FUNCTION_BLOCK conveyor
  (* Standard: 61499-2 *)
  (* Version 0.1, 2017-00-25, hpea485, UOA *)
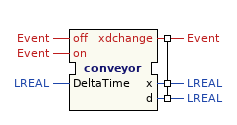
  EVENT_INPUT
    off;
    on;
  END_EVENT
  EVENT_OUTPUT
    xdchange WITH x, d;
  END_EVENT
  VAR_INPUT
    DeltaTime : LREAL := 0.01;
  END_VAR
  VAR_OUTPUT
    x : LREAL;
    d : LREAL;
  END_VAR
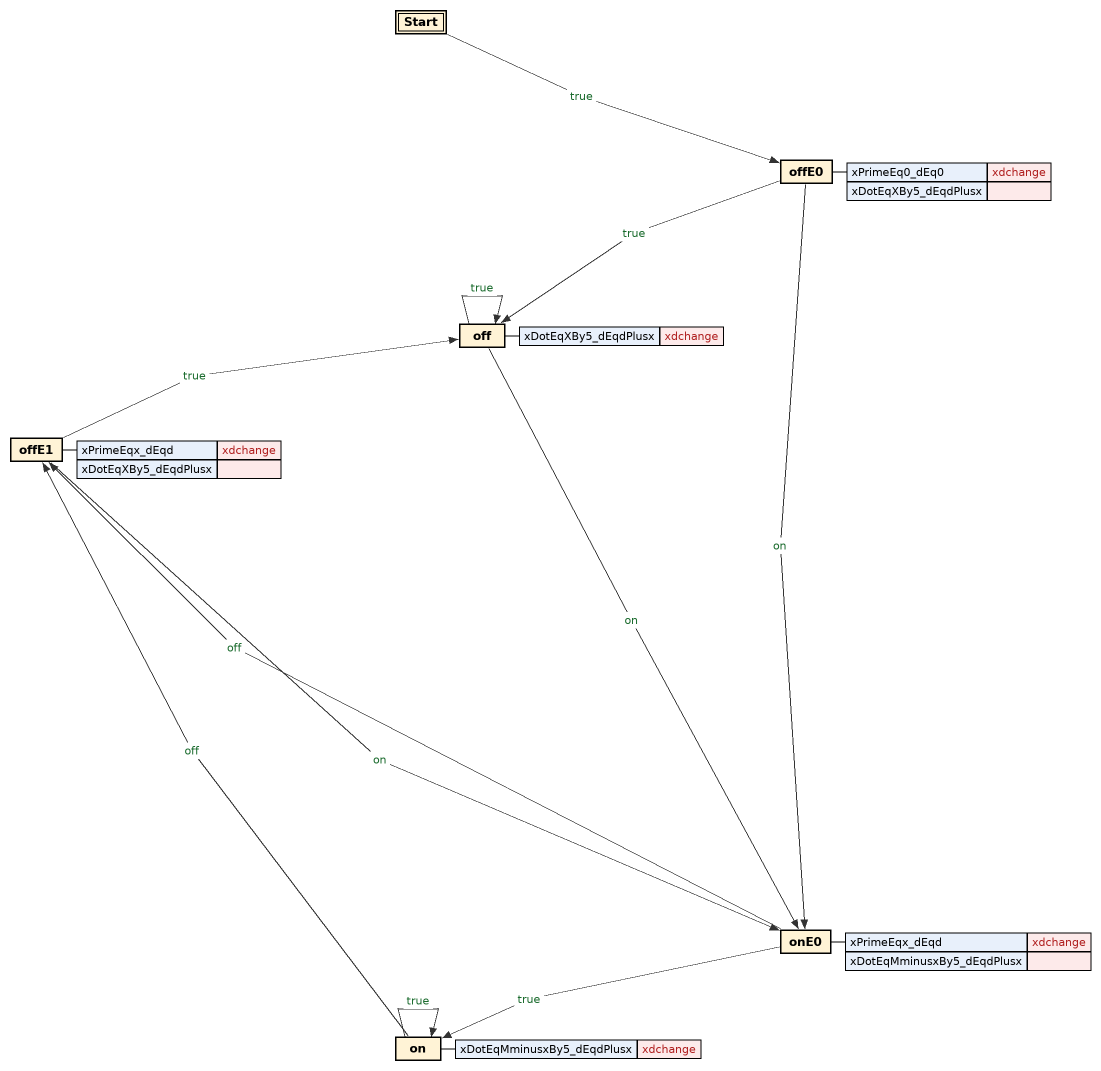
  EC_STATES
    Start;
    offE0 : xPrimeEq0_dEq0 -> xdchange, xDotEqXBy5_dEqdPlusx;
    off : xDotEqXBy5_dEqdPlusx -> xdchange;
    onE0 : xPrimeEqx_dEqd -> xdchange, xDotEqMminusxBy5_dEqdPlusx;
    on : xDotEqMminusxBy5_dEqdPlusx -> xdchange;
    offE1 : xPrimeEqx_dEqd -> xdchange, xDotEqXBy5_dEqdPlusx;
  END_STATES
  EC_TRANSITIONS
    Start TO offE0 := true;
    offE0 TO onE0 := on;
    offE0 TO off := true;
    off TO onE0 := on;
    off TO off := true;
    onE0 TO offE1 := off;
    onE0 TO on := true;
    on TO offE1 := off;
    on TO on := true;
    offE1 TO onE0 := on;
    offE1 TO off := true;
  END_TRANSITIONS
  ALGORITHM xPrimeEq0_dEq0 IN C: (* ODE_init *)
x_prime = 0;
d = 0;
  END_ALGORITHM
  ALGORITHM xPrimeEqx_dEqd IN C: (* ODE_init *)
x_prime = x;
d = d;
  END_ALGORITHM
  ALGORITHM xDotEqXBy5_dEqdPlusx IN C: (* ODE *)
x_dot = x / 5;
d = d + x;
  END_ALGORITHM
  ALGORITHM xDotEqMminusxBy5_dEqdPlusx IN C: (* ODE *)
x_dot = (0.02 - x) / 5;
d = d + x;
  END_ALGORITHM
END_FUNCTION_BLOCK
